{attribute addProperty BoxType "EJ3108-0000-0017"}
{attribute addProperty Id "AI_Standard_ChannelAT %I*ARRAY[0..14] OF AI_Standard_Channel_F16A160D256320WcStateAT %I*WcState_98A4DF7520.250InfoDataAT %I*InfoData_BC63D37F80100"}
{attribute addProperty CRC "1252681791"}
{attribute addProperty SizeInBites "338"}
{attribute addProperty SizeInBytes "42.25"}
TYPE EJ3108_EA60A077 :
STRUCT
	{attribute addProperty Name "AI_Standard_Channel"}
	AI_Standard_Channel : ARRAY[0..14] OF AI_Standard_Channel_F16A160D;
	{attribute addProperty Name "WcState"}
	WcState : WcState_98A4DF75;
	{attribute addProperty Name "InfoData"}
	InfoData : InfoData_BC63D37F;
END_STRUCT
END_TYPE

(* stored: Version 1.2.0.0, ProductVersion 3.1.4024.9
   DUT EJ3108_EA60A077: Id {cf67d515-002b-43e7-b84a-8dd63f7b1701} *)
